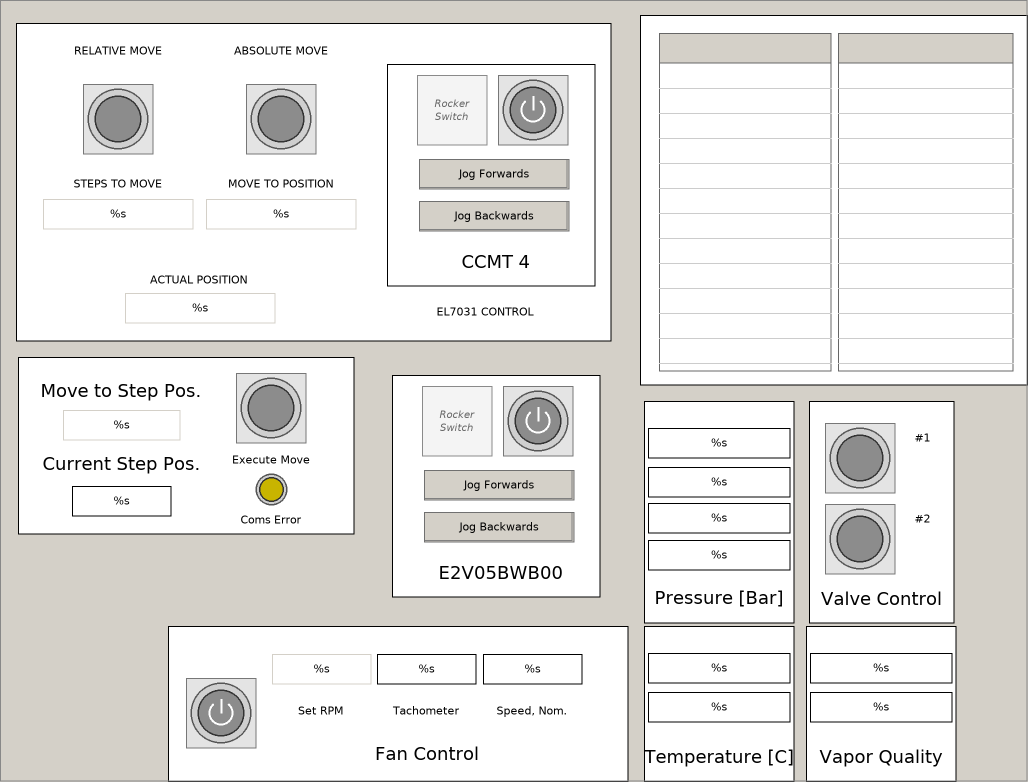
VISUALIZATION Visu_MAIN  // 1028x782
    RoundedRectangle (18,357 336x177)
    Group (392,375 208x222)
        RoundedRectangle (0,0 208x222)
        Button (32,95 150x30), "Jog Forwards"
            tap MAIN.fbAxis2.bJogFwd
        Button (32,137 150x30), "Jog Backwards"
            tap MAIN.fbAxis2.bJogBack
        PowerSwitch (111,11 70x70), variable: MAIN.fbAxis2.bReset, behaviour: TOGGLE, style: Switch-PowerSwitch-Gray
        RockerSwitch (30,11 70x70), variable: MAIN.fbAxis2.bEnable, behaviour: TOGGLE, style: Switch-RockerSwitch-Gray
        Label (34,180 150x36), "E2V05BWB00"
    Group (809,401 145x222)
        RoundedRectangle (0,0 145x222)
        PushSwitchLed (16,22 70x70), variable: bRelay1, behaviour: TOGGLE, style: Switch-PushSwitchLed-Gray
        PushSwitchLed (16,103 70x70), variable: bRelay2, behaviour: TOGGLE, style: Switch-PushSwitchLed-Gray
        Label (7,180 131x36), "Valve Control"
        Label (89,22 49x30), "#1"
        Label (89,103 49x30), "#2"
    Group (644,401 150x222)
        RoundedRectangle (0,0 150x222)
        Label (7,179 136x36), "Pressure [Bar]"
        Rectangle (4,27 142x30), "%s", text variable: MAIN.sPress01
        Rectangle (4,66 142x30), "%s", text variable: MAIN.sPress02
        Rectangle (4,102 142x30), "%s", text variable: MAIN.sPress03
        Rectangle (4,139 142x30), "%s", text variable: MAIN.sPress04
    Group (644,626 150x156)
        RoundedRectangle (0,0 150x156)
        Label (4,113 143x36), "Temperature [C]"
        Rectangle (4,27 142x30), "%s", text variable: MAIN.SurfaceRTD1
        Rectangle (4,66 142x30), "%s", text variable: MAIN.SurfaceRTD2
    Group (806,626 150x156)
        RoundedRectangle (0,0 150x156)
        Label (7,113 136x36), "Vapor Quality"
        Rectangle (4,27 142x30), "%s", text variable: MAIN.sVaporQual
        Rectangle (4,66 142x30), "%s", text variable: MAIN.sPress02
    RoundedRectangle (640,15 388x370)
    Table (659,33 172x338), data array: MAIN.fbFormatRTD.RTDarray
        p3854506369: MAIN.fbFormatRTD.RTDarray[INDEX]
        p2232123230: RTD Temperature
    Table (838,33 175x338), data array: MAIN.fbmVtoTemp.degCtempArray
        p3854506369: MAIN.fbmVtoTemp.degCtempArray[INDEX]
    RoundedRectangle (168,626 460x156)
    Label (359,736 136x36), "Fan Control"
    PowerSwitch (186,678 70x70), variable: MAIN.bFanEnable, behaviour: TOGGLE, style: Switch-PowerSwitch-Gray
    Label (273,693 96x36), "Set RPM"
    Rectangle (377,654 99x30), "%s", text variable: MAIN.Fan1.f_tachometerData
    Label (378,693 96x36), "Tachometer"
    Rectangle (483,654 99x30), "%s", text variable: MAIN.Fan1.f_speedNominal
    Label (484,693 96x36), "Speed, Nom."
    Textfield (272,654 99x30), "%s", text variable: MAIN.smbRPM
        OnMouseDown: write the text variable via Default
    Group (16,23 595x318)
        RoundedRectangle (0,0 595x318)
        Textfield (109,270 150x30), "%s", text variable: MAIN.fbAxis1.fbRead_Position_Axis.Position
            OnMouseDown: write the text variable via Default
        Label (108,242 150x30), "ACTUAL POSITION"
        PushSwitch (67,61 70x70), variable: MAIN.bMoveRelative, behaviour: TOGGLE, style: Switch-PushSwitch-Gray
        Label (27,13 150x30), "RELATIVE MOVE"
        Textfield (27,176 150x30), "%s", text variable: MAIN.sStepperNumSteps
            OnMouseClick: write the text variable via Default
        Label (27,146 150x30), "STEPS TO MOVE"
        Group (190,13 150x118)
            PushSwitch (40,48 70x70), variable: MAIN.bMoveAbsolute, behaviour: TOGGLE, style: Switch-PushSwitch-Gray
            Label (0,0 150x30), "ABSOLUTE MOVE"
        Label (190,146 150x30), "MOVE TO POSITION"
        Textfield (190,176 150x30), "%s", text variable: MAIN.sStepperGoTo
            OnMouseClick: write the text variable via Default
        RoundedRectangle (371,41 208x222)
        Button (403,136 150x30), "Jog Forwards"
            tap MAIN.bJogFwd
        Button (403,178 150x30), "Jog Backwards"
            tap MAIN.bJogBack
        PowerSwitch (482,52 70x70), variable: MAIN.fbAxis1.bResetExe, behaviour: TOGGLE, style: Switch-PowerSwitch-Gray
        RockerSwitch (401,52 70x70), variable: MAIN.fbAxis1.bEnable, behaviour: TOGGLE, style: Switch-RockerSwitch-Gray
        Label (405,221 150x36), "CCMT 4"
    PushSwitch (236,373 70x70), variable: MAIN.btnMbActivate, behaviour: TOGGLE, style: Switch-PushSwitch-Gray
    Label (410,297 150x30), "EL7031 CONTROL"
    Textfield (63,410 117x30), "%s", text variable: MAIN.percentOD
        OnMouseDown: write the text variable via Default
    Rectangle (72,486 99x30), "%s", text variable: MAIN.sCCMTPos
    Label (31,373 180x36), "Move to Step Pos."
    Label (42,446 159x36), "Current Step Pos."
    Lamp1 (251,471 41x37), variable: MAIN.fbCCMT4mb.f_mbErrorFlag, style: Lamp-Lamp1-Yellow
    Label (223,502 96x36), "Coms Error"
    Label (223,442 96x36), "Execute Move"
END_VISUALIZATION

(* stored: Version 1.1.0.1, ProductVersion 3.1.4026.7
   Visu Visu_MAIN: Id {43eabe47-151a-492c-8787-97634dc3bfe7} *)
